TYPE Car :
STRUCT
END_STRUCT
END_TYPE

(* stored: Version 1.1.0.1, ProductVersion 3.1.4024.11
   DUT Car: Id {b782856d-dd73-48a1-86e1-46c5b4d51f2c} *)
